FUNCTION_BLOCK ClockCounterInc
  (* Standard: 61499-2 *)
  (* Version 0.0, 2010-02-06, XPMUser, nxtControl GmbH, Template *)
  (* Compiler header: package fb.rt.cs725;import java.util.*;import java.text.SimpleDateFormat; *)
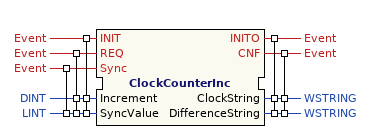
  EVENT_INPUT
    INIT WITH Increment, SyncValue; (* Initialization Request *)
    REQ WITH Increment, SyncValue; (* Normal Execution Request *)
    Sync WITH SyncValue;
  END_EVENT
  EVENT_OUTPUT
    INITO WITH ClockString, DifferenceString; (* Initialization Confirm *)
    CNF WITH ClockString, DifferenceString; (* Execution Confirmation *)
  END_EVENT
  VAR_INPUT
    Increment : DINT; (* Clock * ScaleUpFactor = CLOCK output *)
    SyncValue : LINT;
  END_VAR
  VAR_OUTPUT
    ClockString : WSTRING; (* Output event qualifier *)
    DifferenceString : WSTRING;
  END_VAR
  VAR
    Clock : LINT; (* Output event qualifier *)
    Difference : UDINT;
  END_VAR
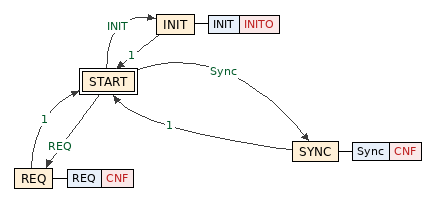
  EC_STATES
    START; (* Initial State *)
    INIT : INIT -> INITO; (* Initialization *)
    REQ : REQ -> CNF; (* Normal execution *)
    SYNC : Sync -> CNF;
  END_STATES
  EC_TRANSITIONS
    START TO INIT := INIT;
    INIT TO START := 1;
    START TO REQ := REQ;
    REQ TO START := 1;
    START TO SYNC := Sync;
    SYNC TO START := 1;
  END_TRANSITIONS
  ALGORITHM INIT IN Java: (* Initialization algorithm *)
Clock.value = new Date().getTime() + SyncValue.value;

// with java.util.Date/Calendar api
Calendar cal = Calendar.getInstance();
cal.setTimeInMillis(Clock.value);

// and here's how to get the String representation
String timeString = new SimpleDateFormat("HH:mm:ss:SSS").format(cal.getTime());

ClockString.value = timeString;
DifferenceString.value = Long.toString(Difference.value);
  END_ALGORITHM
  ALGORITHM REQ IN Java: (* Normally executed algorithm *)
Clock.value = Clock.value + Increment.value;

// with java.util.Date/Calendar api
Calendar cal = Calendar.getInstance();
cal.setTimeInMillis(Clock.value);
// and here's how to get the String representation
String timeString = new SimpleDateFormat("HH:mm:ss:SSS").format(cal.getTime());

ClockString.value = timeString;
  END_ALGORITHM
  ALGORITHM Sync IN ST:
Difference := SyncValue - Clock;
Clock := SyncValue;


System.out.println(Clock + " " + SyncValue);

ClockString := Long.toString(Clock);
DifferenceString := Long.toString(Difference);
  END_ALGORITHM
END_FUNCTION_BLOCK
